(* CoDeSys 2.3.9.48 project: PLC128.pro *)
(* Libraries: SerComm.lib 31.5.11 09:06:48, WagoLibSockets.lib 14.5.12 12:49:54, SysLibSockets.lib 5.5.11 09:22:24, Standard.lib 8.11.10 12:37:48, SYSLIBCALLBACK.LIB 8.11.10 12:37:48, NETVARUDP_LIB_V23.LIB 8.11.10 12:37:48, SysLibCom.lib 8.11.10 12:37:48, Serial_Interface_01.lib 22.4.13 12:50:14 *)

(* PLC configuration (modules and I/O channels)
0750-0652#24 RS-232/RS-485 Interface adjustable (24 Bytes) [Type_30_1_Channels] node 0, in %IB28 out %QB28 {INTTypePAAssignment = PLC; INTTypeModule = plugged}
  AT %IB0 [BYTEOnB_I] First Byte of 24
  AT %QB0 [BYTEOnB_Q] First Byte of 24
0750-0653/0003-0000#03 RS485 Interface (Adjustable), 3 Bytes [Type_21_1_Channels] node 0, in %IB28 out %QB28 {INTTypePAAssignment = PLC; INTTypeModule = plugged}
  AT %IX12.0 [BOOLOnX_I] Transmission acknowledgement
  AT %IX12.1 [BOOLOnX_I] Reception request
  AT %IX12.2 [BOOLOnX_I] Initialization acknowledgement
  AT %IX12.3 [BOOLOnX_I] Input buffer is full
  AT %IX12.4 [BOOLOnX_I] Number of received characters Bit 0
  AT %IX12.5 [BOOLOnX_I] Number of received characters Bit 1
  AT %IX12.6 [BOOLOnX_I] Number of received characters Bit 2
  AT %IB25 [BYTEOnB_I] Input data Byte 0
  AT %IB26 [BYTEOnB_I] Input data Byte 1
  AT %IB27 [BYTEOnB_I] Input data Byte 2
  AT %QX12.0 [BOOLOnX_Q] Transmission request
  AT %QX12.1 [BOOLOnX_Q] Reception acknowledgement
  AT %QX12.2 [BOOLOnX_Q] Initialization request
  AT %QX12.4 [BOOLOnX_Q] Number of characters Bit 0
  AT %QX12.5 [BOOLOnX_Q] Number of characters Bit 1
  AT %QX12.6 [BOOLOnX_Q] Number of characters Bit 2
  AT %QB25 [BYTEOnB_Q] Output data Byte 0
  AT %QB26 [BYTEOnB_Q] Output data Byte 1
  AT %QB27 [BYTEOnB_Q] Output data Byte 2
0750-0653/0003-0000#03 RS485 Interface (Adjustable), 3 Bytes [Type_21_1_Channels] node 0, in %IB52 out %QB52 {INTTypePAAssignment = PLC; INTTypeModule = plugged}
  AT %IX14.0 [BOOLOnX_I] Transmission acknowledgement
  AT %IX14.1 [BOOLOnX_I] Reception request
  AT %IX14.2 [BOOLOnX_I] Initialization acknowledgement
  AT %IX14.3 [BOOLOnX_I] Input buffer is full
  AT %IX14.4 [BOOLOnX_I] Number of received characters Bit 0
  AT %IX14.5 [BOOLOnX_I] Number of received characters Bit 1
  AT %IX14.6 [BOOLOnX_I] Number of received characters Bit 2
  AT %IB29 [BYTEOnB_I] Input data Byte 0
  AT %IB30 [BYTEOnB_I] Input data Byte 1
  AT %IB31 [BYTEOnB_I] Input data Byte 2
  AT %QX14.0 [BOOLOnX_Q] Transmission request
  AT %QX14.1 [BOOLOnX_Q] Reception acknowledgement
  AT %QX14.2 [BOOLOnX_Q] Initialization request
  AT %QX14.4 [BOOLOnX_Q] Number of characters Bit 0
  AT %QX14.5 [BOOLOnX_Q] Number of characters Bit 1
  AT %QX14.6 [BOOLOnX_Q] Number of characters Bit 2
  AT %QB29 [BYTEOnB_Q] Output data Byte 0
  AT %QB30 [BYTEOnB_Q] Output data Byte 1
  AT %QB31 [BYTEOnB_Q] Output data Byte 2
Fieldbus variables [FB_VARS] node 1, in %IB0 out %QB0
fb_var0 AT %ID128 [DWORDOnD_I] DWORD
DWORD, Fieldbus input [FBVAR_DWORD_IN] node 2, in %IB0 out %QB0
  fb_var4 AT %ID129 [DWORDOnD_I] DWORD
DWORD, Fieldbus output [FBVAR_DWORD_OUT] node 3, in %IB0 out %QB0
  fb_var9 AT %QD128 [DWORDOnD_Q] DWORD
DWORD, Fieldbus output [FBVAR_DWORD_OUT] node 4, in %IB0 out %QB0
  fb_var8 AT %QD129 [DWORDOnD_Q] DWORD
DWORD, Fieldbus output [FBVAR_DWORD_OUT] node 5, in %IB0 out %QB0
  fb_var7 AT %QD130 [DWORDOnD_Q] DWORD
DWORD, Fieldbus output [FBVAR_DWORD_OUT] node 6, in %IB0 out %QB0
  fb_var6 AT %QD131 [DWORDOnD_Q] DWORD
DWORD, Fieldbus output [FBVAR_DWORD_OUT] node 7, in %IB0 out %QB0
  fb_var5 AT %QD132 [DWORDOnD_Q] DWORD
DWORD, Fieldbus input [FBVAR_DWORD_IN] node 8, in %IB0 out %QB0
  fb_var3 AT %ID130 [DWORDOnD_I] DWORD
DWORD, Fieldbus input [FBVAR_DWORD_IN] node 9, in %IB0 out %QB0
  fb_var2 AT %ID131 [DWORDOnD_I] DWORD
DWORD, Fieldbus input [FBVAR_DWORD_IN] node 10, in %IB0 out %QB0
  fb_var1 AT %ID132 [DWORDOnD_I] DWORD
Flag variables [FLAG_VARS] node 2, in %IB0 out %QB0
Modbus-Master [MB_MASTER] node 3, in %IB0 out %QB0
*)

(* Task configuration *)
TASK TCPServer (PRIORITY := 1, INTERVAL := T#100ms);
	TCPServer();
END_TASK
TASK Ser2 (PRIORITY := 4, INTERVAL := T#500ms);
	RS485();
END_TASK

(* Global variable list: Networkmanagement implicit Variables UDP *)
VAR_GLOBAL CONSTANT
	USE_NWVARS_UDP : BOOL := FALSE;
	MAX_NetVarItems_UDP	: INT := 0;
	MAX_NetVarPDO_Rx_UDP	: INT := 0;
	MAX_NetVarPDO_Tx_UDP	: INT := 0;
	MAX_NetVarOD_UDP		: INT := 0;
END_VAR
VAR_GLOBAL
	pNetVarItems_UDP		: ARRAY[0..MAX_NetVarItems_UDP] OF NetVarDataItem_UDP;
	pNetVarPDO_Rx_UDP		: ARRAY[0..MAX_NetVarPDO_Rx_UDP] OF NetVarPDO_Rx_UDP;
	pNetVarPDO_Tx_UDP		: ARRAY[0..MAX_NetVarPDO_Tx_UDP] OF NetVarPDO_Tx_UDP;
	pNetVarOD_UDP			: ARRAY[0..MAX_NetVarOD_UDP] OF NetVarSDO_UDP;
	pNetVarPDO_Rx_Diagnosis_UDP : ARRAY[0..MAX_NetVarPDO_Rx_UDP] OF NetVarUDPDiagStruct;
	pNetVarPDO_Tx_Diagnosis_UDP : ARRAY[0..MAX_NetVarPDO_Tx_UDP] OF NetVarUDPDiagStruct;
END_VAR

(* POU TCPServer, ST *)
PROGRAM TCPServer
VAR
	diSocket : DINT := -1;
	iPort : INT:=10000;
	Client : CLIENT_ACCEPT := (diSocket := -1);

	bySend :ARRAY [0..5] OF BYTE;
	byRecv : ARRAY [0..10] OF BYTE;
	ArrayRecv1 : ARRAY[0..10] OF BYTE;
	ArrayRecv2 : ARRAY[0..10] OF BYTE;
	Reply : CLIENT_REPLY;
	bCloseClient: BOOL;
	bActive: BOOL := TRUE;
	test: STRING;
END_VAR
bySend[0] := 1;
bySend[1] := 2;
bySend[2] := 3;
bySend[3] := 4;
bySend[4] := 5;
bySend[5] := 6;

IF bActive THEN
	IF diSocket = -1 THEN
		diSocket := TcpServerOpenSocket(iPort, 10, 0);
	END_IF

	IF  Client.diSocket = -1 THEN
		Client := TcpServerWaitForConnect(diSocket, 1);
	END_IF

	IF  Client.diSocket <> -1 THEN
		TcpSendData(Client.diSocket, ADR(bySend), SIZEOF(bySend), 2);
		TcpReceiveData(Client.diSocket, ADR(byRecv), SIZEOF(byRecv), 4);
		IF byRecv[0] = 49 THEN
			ArrayRecv1 := byRecv;
		ELSE
			ArrayRecv2 := byRecv;
		END_IF
		byRecv[0] := 0;
		bCloseClient := TRUE;
	END_IF

	IF bCloseClient THEN
		bCloseClient := FALSE;
		SysSockClose(diSocket:=Client.diSocket);
		Client.diSocket := -1;
	END_IF
END_IF
END_PROGRAM

(* POU TcpServerOpenSocket, ST *)
FUNCTION TcpServerOpenSocket : DINT
VAR_INPUT
	iPort:INT;						(* Port number *)
	diMaxConnections:DINT;		(* Max possible client connections of the server *)
	diMaxDataSize:DINT;			(* Max size of data to transmitt; if size = 0 default values are used *)
END_VAR
VAR
	diSocket:DINT;
	bResult:BOOL;
	sa:SOCKADDRESS;
	bOptNoDelay:BOOL;
	lOptLinger:SOCKET_LINGER;
END_VAR
diSocket:=SysSockCreate(SOCKET_AF_INET, SOCKET_STREAM, SOCKET_IPPROTO_IP);
IF diSocket <> SOCKET_INVALID THEN
	sa.sin_family:=SOCKET_AF_INET;
	sa.sin_addr:=SOCKET_INADDR_ANY;
	sa.sin_port:=SysSockHtons(iPort);
	bResult:=SysSockBind(diSocket, ADR(sa), SIZEOF(sa));
	IF bResult = FALSE THEN
		diSocket:=SOCKET_INVALID;
	ELSE
		bResult:=SysSockListen(diSocket, diMaxConnections);
		IF bResult = FALSE THEN
			diSocket:=SOCKET_INVALID;
		END_IF
	END_IF
END_IF
TcpServerOpenSocket:=diSocket;
END_FUNCTION

(* POU TcpServerWaitForConnect, ST *)
FUNCTION TcpServerWaitForConnect : CLIENT_ACCEPT
VAR_INPUT
	diServerSocket:DINT;
	diTimeout : DINT;	(* Timeout in seconds *)
END_VAR
VAR
	sa:SOCKADDRESS;
	ia:INADDR;
	diSize:DINT;
	fdRead: SOCKET_FD_SET;
	fdWrite:SOCKET_FD_SET;
	fdExcept:SOCKET_FD_SET;
	tvTimeout:SOCKET_TIMEVAL;
END_VAR
tvTimeout.tv_sec := diTimeout ;
tvTimeout.tv_usec := 0;
fdRead.fd_count := 1;
fdRead.fd_array[0] := diServerSocket;
IF (SysSockSelect(SOCKET_FD_SETSIZE, ADR(fdRead), 0, 0, ADR(tvTimeout)) > 0) THEN
	diSize:=SIZEOF(sa);
	TcpServerWaitForConnect.diSocket:=SysSockAccept(diServerSocket, ADR(sa), ADR(diSize));
	ia.S_addr:=DINT_TO_DWORD(sa.sin_addr);
	SysSockInetNtoa(ia, TcpServerWaitForConnect.stIPAddress, SIZEOF(TcpServerWaitForConnect.stIPAddress));
ELSE
	TcpServerWaitForConnect.diSocket := -1;
END_IF
END_FUNCTION

(* POU TcpSendData, ST *)
FUNCTION TcpSendData : DINT
VAR_INPUT
	diSocket:DINT;		(* Socket Id *)
	pbyData:DWORD;		(* Address of data buffer *)
	diDataSize:DINT;		(* Size of data to send *)
	diTImeout : DINT;		(* Timeout in seconds *)
END_VAR
VAR
	fdWrite:SOCKET_FD_SET;
	tvTimeout:SOCKET_TIMEVAL;
END_VAR
tvTimeout.tv_sec := diTimeout ;
tvTimeout.tv_usec := 0;
fdWrite.fd_count := 1;
fdWrite.fd_array[0] := diSocket;
IF (SysSockSelect(SOCKET_FD_SETSIZE, 0, ADR(fdWrite), 0, ADR(tvTimeout)) > 0) THEN
	TcpSendData:=SysSockSend(diSocket, pbyData, diDataSize, 0);
END_IF
END_FUNCTION

(* POU TcpReceiveData, ST *)
FUNCTION TcpReceiveData : DINT
VAR_INPUT
	diSocket:DINT;		(* Socket Id *)
	pbyData:DWORD;		(* Address of data buffer *)
	diDataSize:DINT;		(* Size of data to send *)
	diTImeout : DINT;		(* Timeout in seconds *)
END_VAR
VAR
	fdRead:SOCKET_FD_SET;
	tvTimeout:SOCKET_TIMEVAL;
END_VAR
tvTimeout.tv_sec := diTimeout ;
tvTimeout.tv_usec := 0;
fdRead.fd_count := 1;
fdRead.fd_array[0] := diSocket;
IF (SysSockSelect(SOCKET_FD_SETSIZE, ADR(fdRead), 0, 0, ADR(tvTimeout)) > 0) THEN
	TcpReceiveData:=SysSockRecv(diSocket, pbyData, diDataSize, 0);
END_IF
END_FUNCTION

(* POU RS485, ST *)
PROGRAM RS485
VAR
	Com485: SERCOMM;
	Start: BOOL;
	ReceiveBuffer : typRing_Buffer;
	index : INT;
	Reset: BOOL;
	OpenPort: BOOL := TRUE;
	RecvString : STRING;
	SendString: STRING;
END_VAR
SendString := 'Ciao';

Com485(
	EN := OpenPort,
	COMPORT := 1,
	BAUDRATE := BAUD_57600,
	BYTESIZE  := BS_8,
	FLOW_CONTROL := NO_FLOW_CONTROL,
	PARITY := PARITY_NO,
	STOPBITS := STOPBITS_1,
	BYTES_TO_DO := LEN(SendString),
	SEND_BUFFER := ADR(SendString),
	RECEIVE_BUFFER := ADR(RecvString)
	);

index := index + 1;
END_PROGRAM

(* POU PLC_PRG, ST *)
PROGRAM PLC_PRG
VAR
END_VAR
%QX2.0 := TRUE;
END_PROGRAM

(* POU Configuration/MODBUS_CONFIGURATION, ST *)
PROGRAM MODBUS_CONFIGURATION        
VAR                                
END_VAR                            
(*                                 
   <?xml version="1.0" encoding="UTF-16" standalone="yes"?>
<network xml_structure_version="1" xml_feature_version="1">
	<generator_settings minRTUTaskCycleTimeMs="5" minEthaskCycleTimeMs="5" ethSlaveMultiplier="0.1" rtuInterfaceMultiplier="0.1" taskGeneration="true"/>
</network>
                              
*)                                 
;                                  
END_PROGRAM

(* POU Program485, CFC *)
PROGRAM Program485
VAR
	COM	:	SERIAL_INTERFACE;
	StartSend	:	BOOL;
	ReceiveBuffer	:	typRING_BUFFER;
	Reset	:	BOOL;
	Text	:	STRING := 'Ciao';
	INFO	: BYTE;
END_VAR
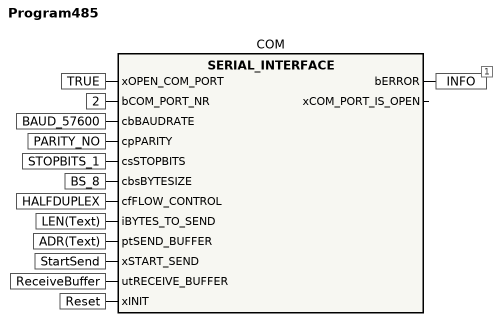
_CFC_ (* Continuous Function Chart, elements in execution order *)
#0 COM:SERIAL_INTERFACE(xOPEN_COM_PORT: TRUE, bCOM_PORT_NR: 2, cbBAUDRATE: BAUD_57600, cpPARITY: PARITY_NO, csSTOPBITS: STOPBITS_1, cbsBYTESIZE: BS_8, cfFLOW_CONTROL: HALFDUPLEX, iBYTES_TO_SEND: LEN(Text), ptSEND_BUFFER: ADR(Text), xSTART_SEND: StartSend, utRECEIVE_BUFFER: ReceiveBuffer, xINIT: Reset)
#1 INFO <= #0.bERROR
_END_CFC_
(* the same logic as Structured Text *)
COM(xOPEN_COM_PORT := TRUE, bCOM_PORT_NR := 2, cbBAUDRATE := BAUD_57600, cpPARITY := PARITY_NO, csSTOPBITS := STOPBITS_1, cbsBYTESIZE := BS_8, cfFLOW_CONTROL := HALFDUPLEX, iBYTES_TO_SEND := LEN(Text), ptSEND_BUFFER := ADR(Text), xSTART_SEND := StartSend, utRECEIVE_BUFFER := ReceiveBuffer, xINIT := Reset);
INFO := COM.bERROR;
END_PROGRAM

(* POU SER485, ST *)
PROGRAM SER485
VAR
(* Communicationparams for 750-65x/003-000 only*)
	wBaudRate : WORD := 5760;
	bDataBits : BYTE := 8;
	bParity : BYTE := 0;
	bFlowControl : BYTE := 4;
	i : INT;
(* COM0 ********************************************)
	COM1 : SERIAL_INTERFACE;
	xOpenPort0 : BOOL := TRUE;
	xInitPort0 : BOOL;
	xSendActive0 : BOOL;
	SendString0 : STRING := 'Msg from COM0';
	ReceiveBuffer0 : typRing_Buffer;
	ReceiveBuffer0OldIndex : INT;
	ReceiveString0 : STRING(255);
	pReceiveStr0 : POINTER TO ARRAY[0..255] OF BYTE;
	ReceiveBytes : BYTE;
	help0Idx : INT;
	iTo2 : INT;
END_VAR
(* Send and Receive for COM0 *)
COM1( bCOM_PORT_NR := 1,
cbBAUDRATE := wBaudRate,
cbsBYTESIZE := bDataBits,
cpPARITY := bParity,
csSTOPBITS := STOPBITS_1,
cfFLOW_CONTROL := bFlowControl,
utRECEIVE_BUFFER := ReceiveBuffer0,
ptSEND_BUFFER := ADR(SendString0),
xINIT := xInitPort0,
xOPEN_COM_PORT := xOpenPort0,
iBYTES_TO_SEND := LEN(SendString0) +1,
xSTART_SEND := xSendActive0 );

(* Display received data for COM0 *)
IF ReceiveBuffer0OldIndex <> ReceiveBuffer0.Index THEN
	iTo2 := ReceiveBuffer0.Index - ReceiveBuffer0OldIndex -1;
	IF iTo2 < 0 THEN
		iTo2 := iTo2 + SIZEOF(ReceiveBuffer0.Data);
	END_IF;
	IF pReceiveStr0 = 0 THEN
		pReceiveStr0 := ADR( ReceiveString0 );
	END_IF;
	FOR i:=0 TO iTo2 DO
		help0Idx := (ReceiveBuffer0OldIndex + i) MOD (SIZEOF(ReceiveBuffer0.Data));
		(*pReceiveStr0^ := ReceiveBuffer0.Data[ help0Idx ];*)
		ReceiveBytes := ReceiveBuffer0.Data[ help0Idx ];
		IF ReceiveBuffer0.Data[ help0Idx ] = 16#00 THEN
			ReceiveBuffer0OldIndex := ReceiveBuffer0.Index;
		END_IF;
	END_FOR;
END_IF;
END_PROGRAM
